{attribute 'qualified_only'}
{attribute 'strict'}
{attribute 'to_string'}
TYPE E_UnitState :
(
    Disabled,
    Idle,
    Ready,
    Running,
    Done,
    Error,
    Aborted
);
END_TYPE

(* stored: Version 1.1.0.1
   DUT E_UnitState: Id {72ad40cf-e9c6-4f3a-b710-def3cb7e9f22} *)
